FUNCTION_BLOCK EL3218
VAR
	_io : EL3xx8_Data;
	{attribute addProperty Name "WcState"}
	_wcState : WcStateInputToggle;
	{attribute addProperty Name "Info data"}
	_infoData : InfoDataAds;
END_VAR

PROPERTY IO : REFERENCE TO EL3xx8_Data
GET
IO REF= _io;
END_GET
END_PROPERTY

PROPERTY WcState : REFERENCE TO WcStateInputToggle
GET
WcState REF= _wcState;
END_GET
END_PROPERTY

END_FUNCTION_BLOCK

(* stored: Version 1.1.0.1, ProductVersion 3.1.4024.9
   POU EL3218: Id {87be4ee5-b2b1-004e-2d75-ee4578d7ea44}, SpecialFunc None
   Property IO: Id {ba4e681b-e923-04e8-1a22-8258ee9043f6}
   Get Get: Id {889757a7-78d1-07a8-002f-a72aa1832184}
   Property WcState: Id {018ace8a-c56d-09f5-0056-7a5480a3b37c}
   Get Get: Id {617fdec9-b091-06e3-2a57-fc37fa10cdee} *)
